{attribute 'qualified_only'}
{attribute 'strict'}
{attribute 'to_string'}
TYPE TRAFFIC_LIGHT_MODE :
(
	OFF,
	NORMAL,
	BLINKING_YELLOW
);
END_TYPE

(* stored: Version 1.1.0.1
   DUT TRAFFIC_LIGHT_MODE: Id {c86efac7-d94a-497b-9cb3-97b5f57e40a3} *)
